// TIA Portal V21 export
DATA_BLOCK "HMI_Settings_DB"   // DB703
{ S7_Optimized_Access := 'TRUE'; DB_Accessible_From_OPC_UA := 'FALSE' }
// stored: AutoNumber false, DBAccessibleFromOPCUA false, DBAccessibleFromWebserver false, InstanceOfName UDT_Settings, InstanceOfType UDT
"UDT_Settings"
   // VAR RETAIN
   //    AlarmDelays : Struct
   //       Protection : Time;
   //       Communication : Time;
   //       DriveFault : Time;
   //       LowCurrent : Time;
   //       WorkConfirmation : Time;
   //       Tank : Time;
   //       Sensor { ExternalAccessible := 'False'; ExternalVisible := 'False'; ExternalWritable := 'False'} : Time;
   //    END_STRUCT;
   //    Sensors : Struct
   //       LiquidLevel : Struct
   //          Tank_1 : "AnalogInputSettings";
   //          Tank_2 : "AnalogInputSettings";
   //       END_STRUCT;
   //    END_STRUCT;
   // END_VAR
BEGIN
END_DATA_BLOCK
